FUNCTION_BLOCK AddCommand EXTENDS CommandBase
VAR_INPUT
	Val1 : REAL;
	Val2 : REAL;
END_VAR
VAR_OUTPUT 
	// The result of the addition command
	Result : REAL;	
END_VAR
VAR
END_VAR

// OO-Class 
;

METHOD PROTECTED Task : BOOL
Result := Val1 + Val2;

// Task comlete;
Task := SUPER^.Task();;
END_METHOD

END_FUNCTION_BLOCK

(* stored: Version 1.1.0.1, ProductVersion 3.1.4022.10
   POU AddCommand: Id {98998d3f-90e1-4abb-9d41-c1c8d9357edf}, SpecialFunc None
   Method Task: Id {72999091-51a2-4b24-b591-51f1ce1d7835} *)
